INTERFACE I_TankController

METHOD ApplyCooling : BOOL
VAR_INPUT
END_VAR
END_METHOD

METHOD CheckSafety : BOOL
VAR_INPUT
END_VAR
END_METHOD

END_INTERFACE

(* stored: Version 1.1.0.1, ProductVersion 3.1.4024.16
   Itf I_TankController: Id {5fed1668-7925-4a0b-906b-e2d258439e71}
   Method ApplyCooling: Id {ac9eb6bc-7866-49ba-90dc-213de6db3b7b}
   Method CheckSafety: Id {f0550787-2f09-410a-a455-bd8a3571d6cd} *)
